SUBAPPLICATION Uebung_229 (* 2 Taster (I1/I2) auf 1 SR-Latch (Last-Wins) via 2x AX_RF_TRIG + AX_SR, Ausgang Q1 *)
  (* Standard: 61499-2; Description: Copyright (c) 2026 Meisterschulen am Ostbahnhof This program and the accompanying materials are made available under the terms of the Eclipse Public License 2.0 which is available at https://www.eclipse.org/legal/epl-2.0/ SPDX-License-Identifier: EPL-2.0 *)
  (* Version 1.0, 2026-09-06, Franz Höpfinger, Meisterschulen am Ostbahnhof, initial API and implementation and/or initial documentation *)
  PACKAGE Uebungen;
  IMPORT logiBUS::io::DI::logiBUS_DI::Input_I1;
  IMPORT logiBUS::io::DI::logiBUS_DI::Input_I2;
  IMPORT logiBUS::io::DQ::logiBUS_DO::Output_Q1;
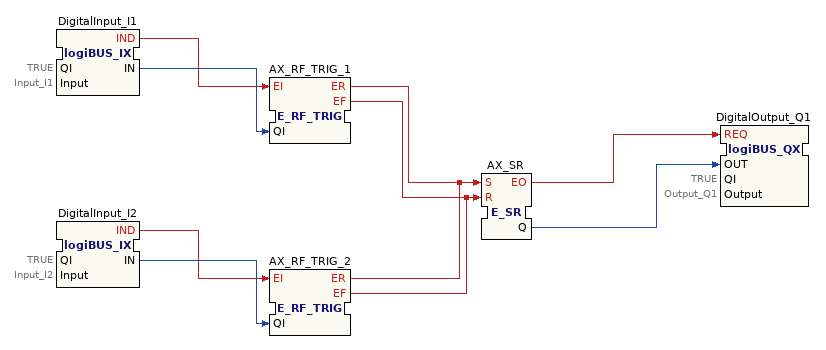
  FBS
    DigitalInput_I1 : logiBUS::io::DI::logiBUS_IX(QI := TRUE, Input := Input_I1);
    DigitalInput_I2 : logiBUS::io::DI::logiBUS_IX(QI := TRUE, Input := Input_I2);
    AX_RF_TRIG_1 : iec61499::events::E_RF_TRIG;
    AX_RF_TRIG_2 : iec61499::events::E_RF_TRIG;
    AX_SR : iec61499::events::E_SR;
    DigitalOutput_Q1 : logiBUS::io::DQ::logiBUS_QX(QI := TRUE, Output := Output_Q1);
  END_FBS
  EVENT_CONNECTIONS
    AX_RF_TRIG_1.ER TO AX_SR.S;
    AX_RF_TRIG_2.ER TO AX_SR.S;
    AX_RF_TRIG_1.EF TO AX_SR.R;
    AX_RF_TRIG_2.EF TO AX_SR.R;
    DigitalInput_I2.IND TO AX_RF_TRIG_2.EI;
    DigitalInput_I1.IND TO AX_RF_TRIG_1.EI;
    AX_SR.EO TO DigitalOutput_Q1.REQ;
  END_CONNECTIONS
  DATA_CONNECTIONS
    DigitalInput_I2.IN TO AX_RF_TRIG_2.QI;
    DigitalInput_I1.IN TO AX_RF_TRIG_1.QI;
    AX_SR.Q TO DigitalOutput_Q1.OUT;
  END_CONNECTIONS
END_SUBAPPLICATION
